{attribute 'GeneratedUsingTerminal: BK1120-0000-0021'}
{attribute addProperty BoxType "BK1120-0000-0021"}
{attribute addProperty Id "Term_381_KL1002KL1002_BB38DA8F0"}
{attribute addProperty CRC "927854571"}
{attribute addProperty Size "0"}
TYPE A_0008_BK1120_0000_0021_374DEFEB EXTENDS BK1120_13409EDF :
STRUCT
	{attribute addProperty Name "Term_381_KL1002"}
	Term_381_KL1002 : KL1002_BB38DA8F;
END_STRUCT
END_TYPE

(* stored: Version 1.2.0.0, ProductVersion 3.1.4024.9
   DUT A_0008_BK1120_0000_0021_374DEFEB: Id {1a7b3e8a-8e39-46e0-89cd-8ecfe8c0d533} *)
